// TIA Portal project "模拟量输入" (V16)

(* hardware
DEVICE "S7-1200 station_1"  S7-1200 Station
   slot 0: "Rack_0"  S7-1200 Rack  Rack  V1.0
   slot 1: "PLC_1"  CPU 1214C DC/DC/Rly  6ES7 214-1HG40-0XB0  V4.4
   slot 2: "AI 4x13BIT/AQ 2x14BIT_1"  SM 1234 AI4/AQ2  6ES7 234-4HE30-0XB0  V1.0
*)

// ===== PLC "PLC_1"  CPU 1214C DC/DC/Rly =====

VAR_GLOBAL   // PLC tag table "默认变量表"
   "Tag_1" AT %IW96 : Int;
   "Tag_2" AT %MD0 : Real;
   "实际工程值" AT %MD4 : Real;
   "Tag_3" AT %MD8 : Real;
   "Tag_4" AT %QW96 : Int;
   "Tag_5" AT %MW12 : Int;
   "传感器感应经过D/A转换的值" AT %IW8 : Int;
   "频率显示" AT %MD34 : Real;
   "下料输送频率显示" AT %MD30 : Real;
   "石灰精密投频率" AT %IW10 : Int;
   "Tag_6" AT %IW12 : Int;
   "Tag_7" AT %MD38 : Real;
   "Tag_8" AT %QD10 : Real;
   "Tag_9" AT %QD14 : Real;
   "Tag_10" AT %QD18 : Real;
END_VAR

DATA_BLOCK "模拟量"   // DB1
{ S7_Optimized_Access := 'TRUE' }
VERSION : 0.1
   VAR
      模拟量输入 : Struct
         中间变换值1 : Real;
         中间变换值2 : Real;
         中间变换值3 : Real;
      END_STRUCT;
      模拟量输出 : Struct
         中间变换值1 : Real;
      END_STRUCT;
   END_VAR
BEGIN
END_DATA_BLOCK

FUNCTION "个路模拟量输入" : Void   // FC1, LAD
{ S7_Optimized_Access := 'TRUE' }
VERSION : 0.1
   VAR_INPUT
      模拟量输入上限 : Int;
      模拟量输入下限 : Int;
      工程值上限 : Real;
      工程值下限 : Real;
      输入值 : Int;
   END_VAR
   VAR_OUTPUT
      输出 : Real;
   END_VAR
BEGIN

REGION Network 1: 模拟量转化为标准值，及百分比
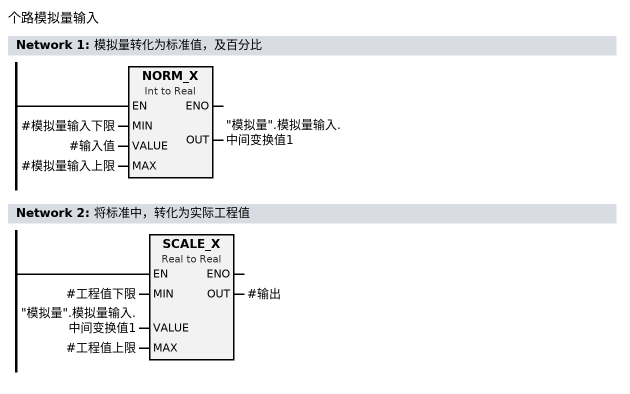
   RUNG wire#powerrail
      { S7_Templates := "[SrcType := Int, DestType := Real]" } Normalize(min := #模拟量输入下限, value := #输入值, max := #模拟量输入上限, out => "模拟量".模拟量输入.中间变换值1)
   END_RUNG
   // the same network as SCL:
   "模拟量".模拟量输入.中间变换值1 := NORM_X(MIN := #模拟量输入下限, VALUE := #输入值, MAX := #模拟量输入上限);
END_REGION

REGION Network 2: 将标准中，转化为实际工程值
   RUNG wire#powerrail
      { S7_Templates := "[SrcType := Real, DestType := Real]" } Scale(min := #工程值下限, value := "模拟量".模拟量输入.中间变换值1, max := #工程值上限, out => #输出)
   END_RUNG
   // the same network as SCL:
   #输出 := SCALE_X(MIN := #工程值下限, VALUE := "模拟量".模拟量输入.中间变换值1, MAX := #工程值上限);
END_REGION
END_FUNCTION

FUNCTION "全部模拟量输入" : Void   // FC2, LAD
{ S7_Optimized_Access := 'TRUE' }
VERSION : 0.1
BEGIN

REGION Network 1
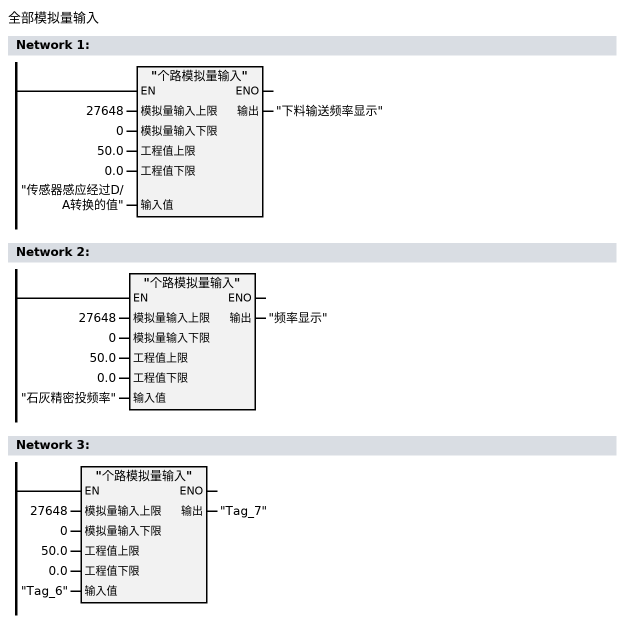
   RUNG wire#powerrail
      "个路模拟量输入"(模拟量输入上限 := 27648, 模拟量输入下限 := 0, 工程值上限 := 50.0, 工程值下限 := 0.0, 输入值 := "传感器感应经过D/A转换的值", 输出 => "下料输送频率显示")
   END_RUNG
   // the same network as SCL:
   "个路模拟量输入"(模拟量输入上限 := 27648,
             模拟量输入下限 := 0,
             工程值上限 := 50.0,
             工程值下限 := 0.0,
             输入值 := "传感器感应经过D/A转换的值",
             输出 => "下料输送频率显示");
END_REGION

REGION Network 2
   RUNG wire#powerrail
      "个路模拟量输入"(模拟量输入上限 := 27648, 模拟量输入下限 := 0, 工程值上限 := 50.0, 工程值下限 := 0.0, 输入值 := "石灰精密投频率", 输出 => "频率显示")
   END_RUNG
   // the same network as SCL:
   "个路模拟量输入"(模拟量输入上限 := 27648, 模拟量输入下限 := 0, 工程值上限 := 50.0, 工程值下限 := 0.0, 输入值 := "石灰精密投频率", 输出 => "频率显示");
END_REGION

REGION Network 3
   RUNG wire#powerrail
      "个路模拟量输入"(模拟量输入上限 := 27648, 模拟量输入下限 := 0, 工程值上限 := 50.0, 工程值下限 := 0.0, 输入值 := "Tag_6", 输出 => "Tag_7")
   END_RUNG
   // the same network as SCL:
   "个路模拟量输入"(模拟量输入上限 := 27648, 模拟量输入下限 := 0, 工程值上限 := 50.0, 工程值下限 := 0.0, 输入值 := "Tag_6", 输出 => "Tag_7");
END_REGION
END_FUNCTION

FUNCTION "个路模拟量输出" : Void   // FC3, LAD
{ S7_Optimized_Access := 'TRUE' }
VERSION : 0.1
   VAR_INPUT
      工程值上限 : Real;
      工程值下限 : Real;
      "电压/电流标准值上限" : Real;
      "电压/电流标准值下限" : Real;
      输入 : Real;
   END_VAR
   VAR_OUTPUT
      输出 : Real;
   END_VAR
BEGIN

REGION Network 1
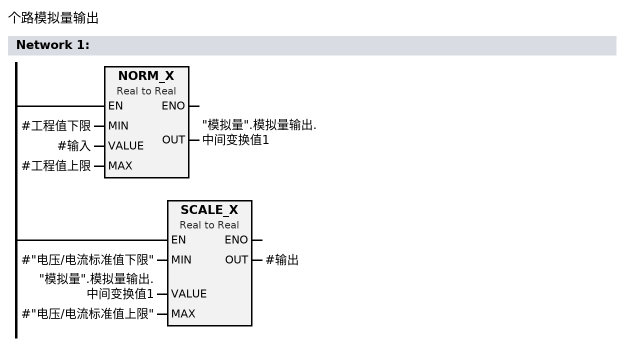
   RUNG wire#powerrail
      { S7_Templates := "[SrcType := Real, DestType := Real]" } Normalize(min := #工程值下限, value := #输入, max := #工程值上限, out => "模拟量".模拟量输出.中间变换值1)
   END_RUNG
   RUNG wire#powerrail
      { S7_Templates := "[SrcType := Real, DestType := Real]" } Scale(min := #"电压/电流标准值下限", value := "模拟量".模拟量输出.中间变换值1, max := #"电压/电流标准值上限", out => #输出)
   END_RUNG
   // the same network as SCL:
   "模拟量".模拟量输出.中间变换值1 := NORM_X(MIN := #工程值下限, VALUE := #输入, MAX := #工程值上限);
   #输出 := SCALE_X(MIN := #"电压/电流标准值下限", VALUE := "模拟量".模拟量输出.中间变换值1, MAX := #"电压/电流标准值上限");
END_REGION
END_FUNCTION

FUNCTION "模拟量输出" : Void   // FC4, LAD
{ S7_Optimized_Access := 'TRUE' }
VERSION : 0.1
BEGIN

REGION Network 1
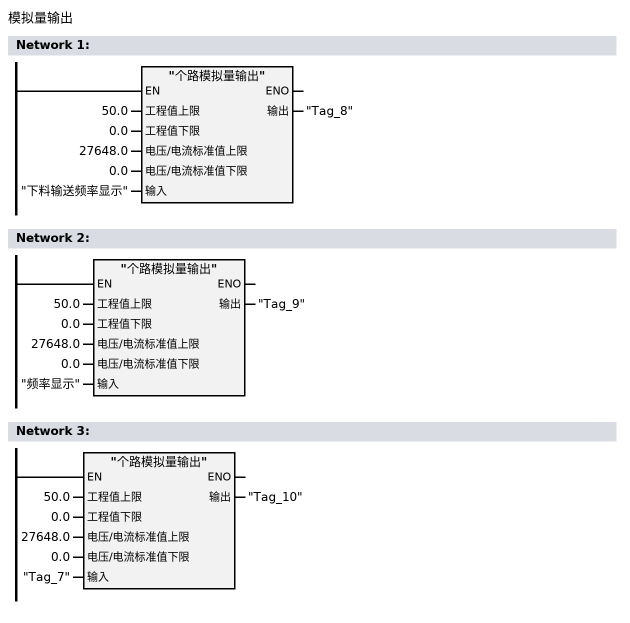
   RUNG wire#powerrail
      "个路模拟量输出"(工程值上限 := 50.0, 工程值下限 := 0.0, "电压/电流标准值上限" := 27648.0, "电压/电流标准值下限" := 0.0, 输入 := "下料输送频率显示", 输出 => "Tag_8")
   END_RUNG
   // the same network as SCL:
   "个路模拟量输出"(工程值上限 := 50.0,
             工程值下限 := 0.0,
             "电压/电流标准值上限" := 27648.0,
             "电压/电流标准值下限" := 0.0,
             输入 := "下料输送频率显示",
             输出 => "Tag_8");
END_REGION

REGION Network 2
   RUNG wire#powerrail
      "个路模拟量输出"(工程值上限 := 50.0, 工程值下限 := 0.0, "电压/电流标准值上限" := 27648.0, "电压/电流标准值下限" := 0.0, 输入 := "频率显示", 输出 => "Tag_9")
   END_RUNG
   // the same network as SCL:
   "个路模拟量输出"(工程值上限 := 50.0,
             工程值下限 := 0.0,
             "电压/电流标准值上限" := 27648.0,
             "电压/电流标准值下限" := 0.0,
             输入 := "频率显示",
             输出 => "Tag_9");
END_REGION

REGION Network 3
   RUNG wire#powerrail
      "个路模拟量输出"(工程值上限 := 50.0, 工程值下限 := 0.0, "电压/电流标准值上限" := 27648.0, "电压/电流标准值下限" := 0.0, 输入 := "Tag_7", 输出 => "Tag_10")
   END_RUNG
   // the same network as SCL:
   "个路模拟量输出"(工程值上限 := 50.0,
             工程值下限 := 0.0,
             "电压/电流标准值上限" := 27648.0,
             "电压/电流标准值下限" := 0.0,
             输入 := "Tag_7",
             输出 => "Tag_10");
END_REGION
END_FUNCTION

ORGANIZATION_BLOCK "Main"   // OB1, LAD, ProgramCycle
TITLE = "Main Program Sweep (Cycle)"
{ S7_Optimized_Access := 'TRUE' }
VERSION : 0.1
   VAR_INPUT
      Initial_Call : Bool;   // Initial call of this OB
      Remanence : Bool;   // =True, if remanent data are available
   END_VAR
BEGIN

REGION Network 1: 先将传感器传过来，通过A/D转换后的，数值，转换成百分比
   // 在AI模块中模拟量输入通道0接0-20mA的电流信号，通道0的地址是iw96
   // 对应实际工程值，程序转换如下，先把iw112测出来的模拟值对应到0-27648，
   // 转换成百分比放到MOD中
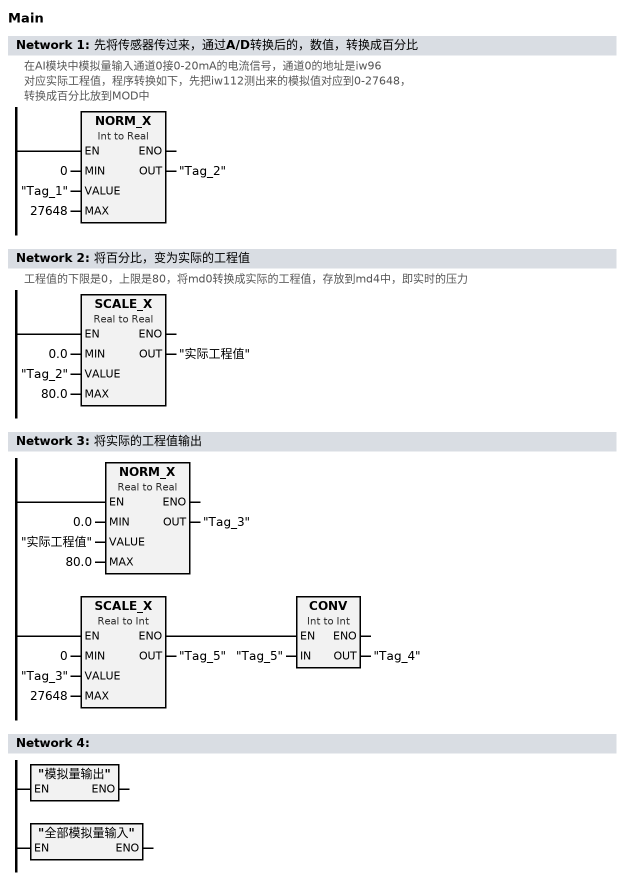
   RUNG wire#powerrail
      { S7_Templates := "[SrcType := Int, DestType := Real]" } Normalize(min := 0, value := "Tag_1", max := 27648, out => "Tag_2")
   END_RUNG
   // the same network as SCL:
   "Tag_2" := NORM_X(MIN := 0, VALUE := "Tag_1", MAX := 27648);
END_REGION

REGION Network 2: 将百分比，变为实际的工程值
   // 工程值的下限是0，上限是80，将md0转换成实际的工程值，存放到md4中，即实时的压力
   RUNG wire#powerrail
      { S7_Templates := "[SrcType := Real, DestType := Real]" } Scale(min := 0.0, value := "Tag_2", max := 80.0, out => "实际工程值")
   END_RUNG
   // the same network as SCL:
   "实际工程值" := SCALE_X(MIN := 0.0, VALUE := "Tag_2", MAX := 80.0);
END_REGION

REGION Network 3: 将实际的工程值输出
   RUNG wire#powerrail
      { S7_Templates := "[SrcType := Real, DestType := Real]" } Normalize(min := 0.0, value := "实际工程值", max := 80.0, out => "Tag_3")
   END_RUNG
   RUNG wire#powerrail
      { S7_Templates := "[SrcType := Real, DestType := Int]" } Scale(min := 0, value := "Tag_3", max := 27648, out => "Tag_5")
      { S7_Templates := "[SrcType := Int, DestType := Int]" } Convert(in := "Tag_5", out => "Tag_4")
   END_RUNG
   // the same network as SCL:
   "Tag_3" := NORM_X(MIN := 0.0, VALUE := "实际工程值", MAX := 80.0);
   "Tag_5" := SCALE_X(MIN := 0, VALUE := "Tag_3", MAX := 27648);
   "Tag_4" := INT_TO_INT("Tag_5");
END_REGION

REGION Network 4
   RUNG wire#powerrail
      "模拟量输出"()
   END_RUNG
   RUNG wire#powerrail
      "全部模拟量输入"()
   END_RUNG
   // the same network as SCL:
   "模拟量输出"();
   "全部模拟量输入"();
END_REGION
END_ORGANIZATION_BLOCK